Universal Robots PolyScope program: brazo_final.urp

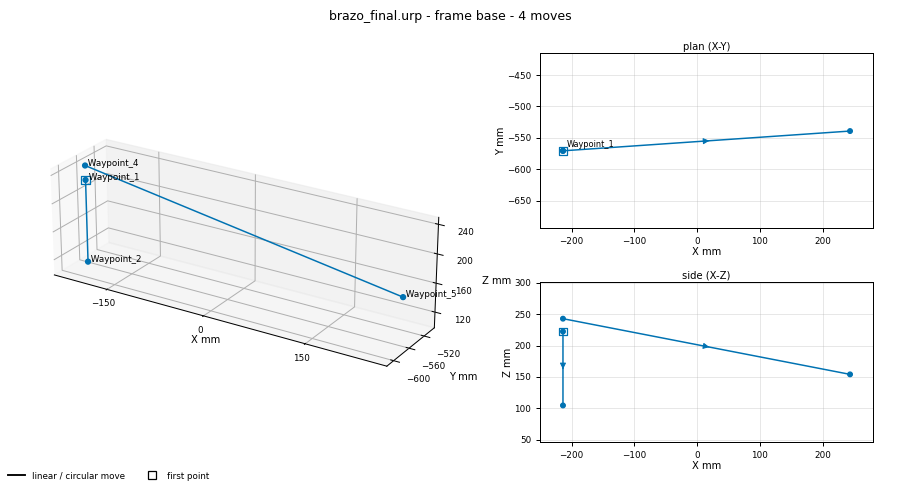
[picture p0: tool path of brazo_final.urp in frame base, 4 of 5 moves have a stored position in this frame; points joined in program order, loops and branches not executed]
Program brazo_final (installation=default directory=/programs/usbdisk/brazo_final createdIn=5.13.0 lastSavedIn=5.13.0 robotSerialNumber=20205500280)
Calibrated DH parameters: a=[0.000126, -0.227628, -0.392536, 0.000072, 0.000053, 0]; d=[0.16267, 78.773992, -78.210517, -0.430145, 0.099656, 0.099678]; alpha=[1.568545, -0.004566, 0.00572, 1.569931, -1.57104, 0]; deltaTheta=[0, -1.006608, 7.298003, -0.008206, 0.000004, 0]
InitVariablesNode
Robot Program (runOnlyOnce=false)
  MoveJ speed 60 deg/s, acceleration 80 deg/s^2 (useActiveTCP=true) feature=Base
    Waypoint Waypoint_1: motionParameters(jointSpeed=3.141593 jointAcceleration=1.396263 cartesianSpeed=0.25 cartesianAcceleration=1.2); TCP in base x=-213.711 y=-570.525 z=222.383 mm, rx=-3.1335 ry=-0.0007 rz=-0.0859 rad; joints [55.344, -74.77, 76.656, -89.796, -87.264, -34.482] deg; TCP offset x=0 y=0 z=234.35 mm, rx=0 ry=0 rz=-3.1416 rad
  URCap RG6 (RG - On Robot, OnRobot A/S) dataModel(depthCompensate=false, force=120, payload=0.0, width=-3, name=RG6(-3))
  MoveL speed 250 mm/s, acceleration 1200 mm/s^2 (useActiveTCP=true) feature=Base
    Waypoint Waypoint_2: motionParameters(jointSpeed=1.047198 jointAcceleration=1.396263 cartesianSpeed=0.25 cartesianAcceleration=1.2); TCP in base x=-213.712 y=-570.557 z=104.626 mm, rx=-3.1336 ry=-0.0007 rz=-0.0857 rad; joints [55.335, -71.918, 90.439, -106.446, -87.287, -34.387] deg
    MoveDirectionNode (selectedDirection=ZMinus toolParams=0.05, 1.2)
      Until TOOL_CONTACT_DETECTION (allowActions=true retraction=0.0125 decelerationAcceleration=3 decelerationAngularAcceleration=34.906585)
        URCap RG6 (RG - On Robot, OnRobot A/S) dataModel(depthCompensate=false, force=120, payload=0.0, width=93, name=RG6(93))
    Waypoint Waypoint_3 (Relative): motionParameters(jointSpeed=1.047198 jointAcceleration=1.396263 cartesianSpeed=0.1 cartesianAcceleration=1.2); relativeFromPosition TCP in base x=-213.687 y=-570.632 z=99.426 mm, rx=-3.1338 ry=-0.0009 rz=-0.0856 rad; joints [55.339, -71.688, 90.932, -107.178, -87.287, -34.386] deg; TCP in base x=-213.715 y=-570.645 z=71.151 mm, rx=-3.1338 ry=-0.0008 rz=-0.0856 rad; joints [55.335, -70.301, 93.452, -111.086, -87.3, -34.363] deg
    URCap RG6 (RG - On Robot, OnRobot A/S) dataModel(depthCompensate=false, force=120, payload=0.0, width=50, name=RG6(50))
    Waypoint Waypoint_4: motionParameters(jointSpeed=1.047198 jointAcceleration=1.396263 cartesianSpeed=0.35 cartesianAcceleration=1.2); TCP in base x=-213.715 y=-570.603 z=242.838 mm, rx=-3.1338 ry=-0.0008 rz=-0.0855 rad; joints [55.35, -74.801, 73.715, -86.844, -87.265, -34.496] deg
    Waypoint Waypoint_5: motionParameters(jointSpeed=1.047198 jointAcceleration=1.396263 cartesianSpeed=0.35 cartesianAcceleration=1.2); TCP in base x=243.533 y=-539.12 z=154.146 mm, rx=-3.1337 ry=-0.0009 rz=-0.0855 rad; joints [99.303, -77.826, 91.145, -103.474, -86.477, 9.587] deg
    URCap RG6 (RG - On Robot, OnRobot A/S) dataModel(depthCompensate=false, force=120, payload=0.0, width=95, name=RG6(95))
